REGION Network 138: Step[3090] : Job[21] Step End
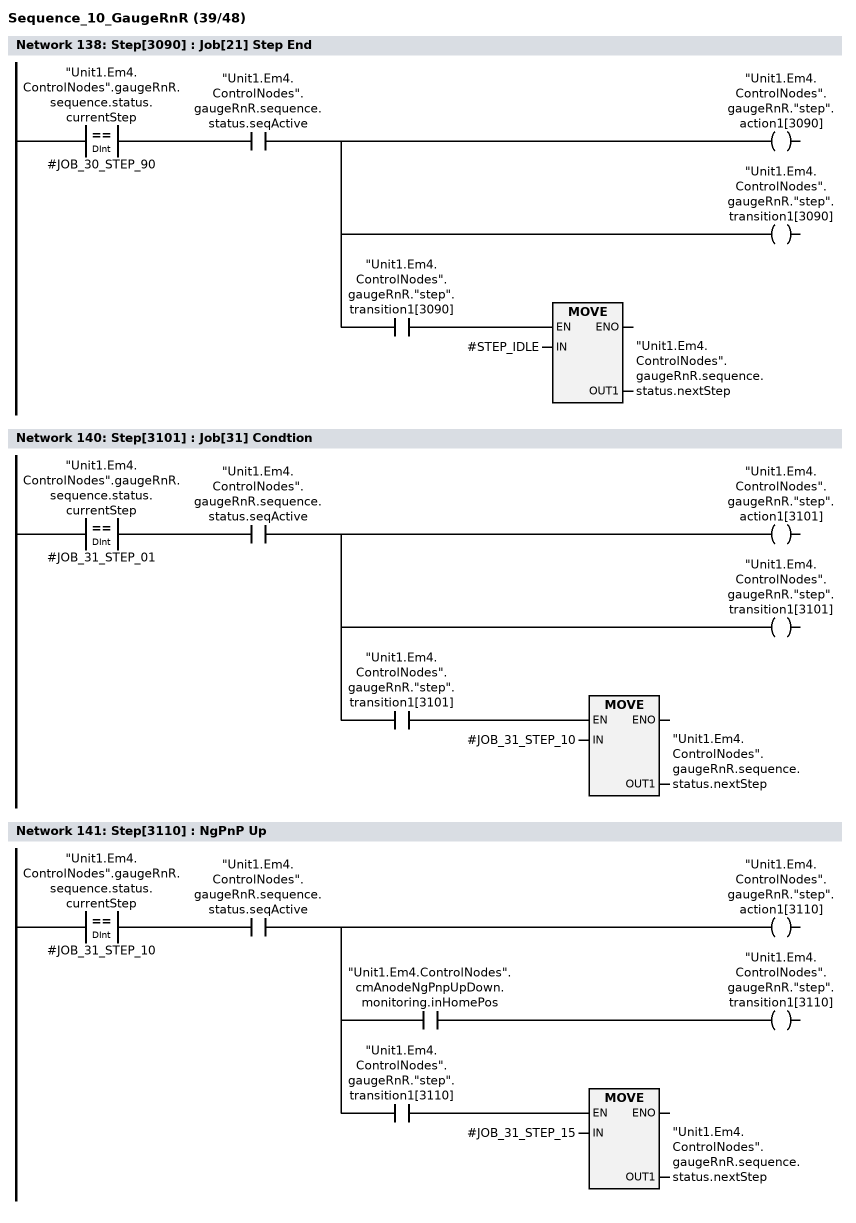
   RUNG wire#powerrail
      { S7_Templates := "SrcType := DInt" } EQ_Contact(in1 := "Unit1.Em4.ControlNodes".gaugeRnR.sequence.status.currentStep, in2 := #JOB_30_STEP_90)
      Contact( "Unit1.Em4.ControlNodes".gaugeRnR.sequence.status.seqActive )
      wire#w1
      Coil( "Unit1.Em4.ControlNodes".gaugeRnR."step".action1[3090] )
   END_RUNG
   RUNG wire#w1
      Coil( "Unit1.Em4.ControlNodes".gaugeRnR."step".transition1[3090] )
   END_RUNG
   RUNG wire#w1
      Contact( "Unit1.Em4.ControlNodes".gaugeRnR."step".transition1[3090] )
      Move(in := #STEP_IDLE, out1 => "Unit1.Em4.ControlNodes".gaugeRnR.sequence.status.nextStep)
   END_RUNG
   // the same network as SCL:
   "Unit1.Em4.ControlNodes".gaugeRnR."step".action1[3090] := ("Unit1.Em4.ControlNodes".gaugeRnR.sequence.status.currentStep = #JOB_30_STEP_90) AND "Unit1.Em4.ControlNodes".gaugeRnR.sequence.status.seqActive;
   "Unit1.Em4.ControlNodes".gaugeRnR."step".transition1[3090] := ("Unit1.Em4.ControlNodes".gaugeRnR.sequence.status.currentStep = #JOB_30_STEP_90) AND "Unit1.Em4.ControlNodes".gaugeRnR.sequence.status.seqActive;
   IF ("Unit1.Em4.ControlNodes".gaugeRnR.sequence.status.currentStep = #JOB_30_STEP_90) AND "Unit1.Em4.ControlNodes".gaugeRnR.sequence.status.seqActive AND "Unit1.Em4.ControlNodes".gaugeRnR."step".transition1[3090] THEN
       "Unit1.Em4.ControlNodes".gaugeRnR.sequence.status.nextStep := #STEP_IDLE;
   END_IF;
END_REGION

REGION Network 139: *************** JOB[31] NG PnP Load MasterPiece ************************
END_REGION

REGION Network 140: Step[3101] : Job[31] Condtion
   RUNG wire#powerrail
      { S7_Templates := "SrcType := DInt" } EQ_Contact(in1 := "Unit1.Em4.ControlNodes".gaugeRnR.sequence.status.currentStep, in2 := #JOB_31_STEP_01)
      Contact( "Unit1.Em4.ControlNodes".gaugeRnR.sequence.status.seqActive )
      wire#w1
      Coil( "Unit1.Em4.ControlNodes".gaugeRnR."step".action1[3101] )
   END_RUNG
   RUNG wire#w1
      Coil( "Unit1.Em4.ControlNodes".gaugeRnR."step".transition1[3101] )
   END_RUNG
   RUNG wire#w1
      Contact( "Unit1.Em4.ControlNodes".gaugeRnR."step".transition1[3101] )
      Move(in := #JOB_31_STEP_10, out1 => "Unit1.Em4.ControlNodes".gaugeRnR.sequence.status.nextStep)
   END_RUNG
   // the same network as SCL:
   "Unit1.Em4.ControlNodes".gaugeRnR."step".action1[3101] := ("Unit1.Em4.ControlNodes".gaugeRnR.sequence.status.currentStep = #JOB_31_STEP_01) AND "Unit1.Em4.ControlNodes".gaugeRnR.sequence.status.seqActive;
   "Unit1.Em4.ControlNodes".gaugeRnR."step".transition1[3101] := ("Unit1.Em4.ControlNodes".gaugeRnR.sequence.status.currentStep = #JOB_31_STEP_01) AND "Unit1.Em4.ControlNodes".gaugeRnR.sequence.status.seqActive;
   IF ("Unit1.Em4.ControlNodes".gaugeRnR.sequence.status.currentStep = #JOB_31_STEP_01) AND "Unit1.Em4.ControlNodes".gaugeRnR.sequence.status.seqActive AND "Unit1.Em4.ControlNodes".gaugeRnR."step".transition1[3101] THEN
       "Unit1.Em4.ControlNodes".gaugeRnR.sequence.status.nextStep := #JOB_31_STEP_10;
   END_IF;
END_REGION

REGION Network 141: Step[3110] : NgPnP Up
   RUNG wire#powerrail
      { S7_Templates := "SrcType := DInt" } EQ_Contact(in1 := "Unit1.Em4.ControlNodes".gaugeRnR.sequence.status.currentStep, in2 := #JOB_31_STEP_10)
      Contact( "Unit1.Em4.ControlNodes".gaugeRnR.sequence.status.seqActive )
      wire#w1
      Coil( "Unit1.Em4.ControlNodes".gaugeRnR."step".action1[3110] )
   END_RUNG
   RUNG wire#w1
      Contact( "Unit1.Em4.ControlNodes".cmAnodeNgPnpUpDown.monitoring.inHomePos )
      Coil( "Unit1.Em4.ControlNodes".gaugeRnR."step".transition1[3110] )
   END_RUNG
   RUNG wire#w1
      Contact( "Unit1.Em4.ControlNodes".gaugeRnR."step".transition1[3110] )
      Move(in := #JOB_31_STEP_15, out1 => "Unit1.Em4.ControlNodes".gaugeRnR.sequence.status.nextStep)
   END_RUNG
   // the same network as SCL:
   "Unit1.Em4.ControlNodes".gaugeRnR."step".action1[3110] := ("Unit1.Em4.ControlNodes".gaugeRnR.sequence.status.currentStep = #JOB_31_STEP_10) AND "Unit1.Em4.ControlNodes".gaugeRnR.sequence.status.seqActive;
   "Unit1.Em4.ControlNodes".gaugeRnR."step".transition1[3110] := ("Unit1.Em4.ControlNodes".gaugeRnR.sequence.status.currentStep = #JOB_31_STEP_10) AND "Unit1.Em4.ControlNodes".gaugeRnR.sequence.status.seqActive AND "Unit1.Em4.ControlNodes".cmAnodeNgPnpUpDown.monitoring.inHomePos;
   IF ("Unit1.Em4.ControlNodes".gaugeRnR.sequence.status.currentStep = #JOB_31_STEP_10) AND "Unit1.Em4.ControlNodes".gaugeRnR.sequence.status.seqActive AND "Unit1.Em4.ControlNodes".gaugeRnR."step".transition1[3110] THEN
       "Unit1.Em4.ControlNodes".gaugeRnR.sequence.status.nextStep := #JOB_31_STEP_15;
   END_IF;
END_REGION

REGION Network 142: Step[3115] : NgPnP 1st Forward
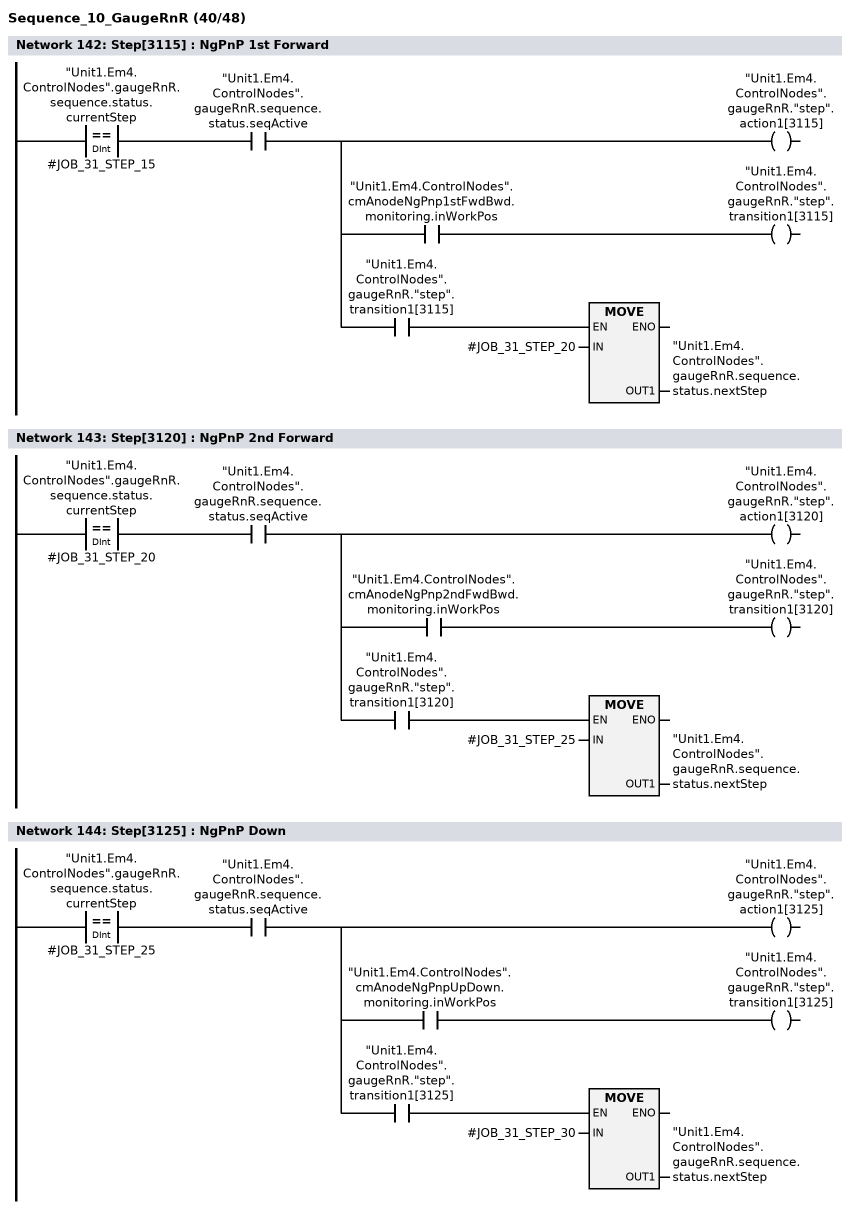
   RUNG wire#powerrail
      { S7_Templates := "SrcType := DInt" } EQ_Contact(in1 := "Unit1.Em4.ControlNodes".gaugeRnR.sequence.status.currentStep, in2 := #JOB_31_STEP_15)
      Contact( "Unit1.Em4.ControlNodes".gaugeRnR.sequence.status.seqActive )
      wire#w1
      Coil( "Unit1.Em4.ControlNodes".gaugeRnR."step".action1[3115] )
   END_RUNG
   RUNG wire#w1
      Contact( "Unit1.Em4.ControlNodes".cmAnodeNgPnp1stFwdBwd.monitoring.inWorkPos )
      Coil( "Unit1.Em4.ControlNodes".gaugeRnR."step".transition1[3115] )
   END_RUNG
   RUNG wire#w1
      Contact( "Unit1.Em4.ControlNodes".gaugeRnR."step".transition1[3115] )
      Move(in := #JOB_31_STEP_20, out1 => "Unit1.Em4.ControlNodes".gaugeRnR.sequence.status.nextStep)
   END_RUNG
   // the same network as SCL:
   "Unit1.Em4.ControlNodes".gaugeRnR."step".action1[3115] := ("Unit1.Em4.ControlNodes".gaugeRnR.sequence.status.currentStep = #JOB_31_STEP_15) AND "Unit1.Em4.ControlNodes".gaugeRnR.sequence.status.seqActive;
   "Unit1.Em4.ControlNodes".gaugeRnR."step".transition1[3115] := ("Unit1.Em4.ControlNodes".gaugeRnR.sequence.status.currentStep = #JOB_31_STEP_15) AND "Unit1.Em4.ControlNodes".gaugeRnR.sequence.status.seqActive AND "Unit1.Em4.ControlNodes".cmAnodeNgPnp1stFwdBwd.monitoring.inWorkPos;
   IF ("Unit1.Em4.ControlNodes".gaugeRnR.sequence.status.currentStep = #JOB_31_STEP_15) AND "Unit1.Em4.ControlNodes".gaugeRnR.sequence.status.seqActive AND "Unit1.Em4.ControlNodes".gaugeRnR."step".transition1[3115] THEN
       "Unit1.Em4.ControlNodes".gaugeRnR.sequence.status.nextStep := #JOB_31_STEP_20;
   END_IF;
END_REGION

REGION Network 143: Step[3120] : NgPnP 2nd Forward
   RUNG wire#powerrail
      { S7_Templates := "SrcType := DInt" } EQ_Contact(in1 := "Unit1.Em4.ControlNodes".gaugeRnR.sequence.status.currentStep, in2 := #JOB_31_STEP_20)
      Contact( "Unit1.Em4.ControlNodes".gaugeRnR.sequence.status.seqActive )
      wire#w1
      Coil( "Unit1.Em4.ControlNodes".gaugeRnR."step".action1[3120] )
   END_RUNG
   RUNG wire#w1
      Contact( "Unit1.Em4.ControlNodes".cmAnodeNgPnp2ndFwdBwd.monitoring.inWorkPos )
      Coil( "Unit1.Em4.ControlNodes".gaugeRnR."step".transition1[3120] )
   END_RUNG
   RUNG wire#w1
      Contact( "Unit1.Em4.ControlNodes".gaugeRnR."step".transition1[3120] )
      Move(in := #JOB_31_STEP_25, out1 => "Unit1.Em4.ControlNodes".gaugeRnR.sequence.status.nextStep)
   END_RUNG
   // the same network as SCL:
   "Unit1.Em4.ControlNodes".gaugeRnR."step".action1[3120] := ("Unit1.Em4.ControlNodes".gaugeRnR.sequence.status.currentStep = #JOB_31_STEP_20) AND "Unit1.Em4.ControlNodes".gaugeRnR.sequence.status.seqActive;
   "Unit1.Em4.ControlNodes".gaugeRnR."step".transition1[3120] := ("Unit1.Em4.ControlNodes".gaugeRnR.sequence.status.currentStep = #JOB_31_STEP_20) AND "Unit1.Em4.ControlNodes".gaugeRnR.sequence.status.seqActive AND "Unit1.Em4.ControlNodes".cmAnodeNgPnp2ndFwdBwd.monitoring.inWorkPos;
   IF ("Unit1.Em4.ControlNodes".gaugeRnR.sequence.status.currentStep = #JOB_31_STEP_20) AND "Unit1.Em4.ControlNodes".gaugeRnR.sequence.status.seqActive AND "Unit1.Em4.ControlNodes".gaugeRnR."step".transition1[3120] THEN
       "Unit1.Em4.ControlNodes".gaugeRnR.sequence.status.nextStep := #JOB_31_STEP_25;
   END_IF;
END_REGION

REGION Network 144: Step[3125] : NgPnP Down
   RUNG wire#powerrail
      { S7_Templates := "SrcType := DInt" } EQ_Contact(in1 := "Unit1.Em4.ControlNodes".gaugeRnR.sequence.status.currentStep, in2 := #JOB_31_STEP_25)
      Contact( "Unit1.Em4.ControlNodes".gaugeRnR.sequence.status.seqActive )
      wire#w1
      Coil( "Unit1.Em4.ControlNodes".gaugeRnR."step".action1[3125] )
   END_RUNG
   RUNG wire#w1
      Contact( "Unit1.Em4.ControlNodes".cmAnodeNgPnpUpDown.monitoring.inWorkPos )
      Coil( "Unit1.Em4.ControlNodes".gaugeRnR."step".transition1[3125] )
   END_RUNG
   RUNG wire#w1
      Contact( "Unit1.Em4.ControlNodes".gaugeRnR."step".transition1[3125] )
      Move(in := #JOB_31_STEP_30, out1 => "Unit1.Em4.ControlNodes".gaugeRnR.sequence.status.nextStep)
   END_RUNG
   // the same network as SCL:
   "Unit1.Em4.ControlNodes".gaugeRnR."step".action1[3125] := ("Unit1.Em4.ControlNodes".gaugeRnR.sequence.status.currentStep = #JOB_31_STEP_25) AND "Unit1.Em4.ControlNodes".gaugeRnR.sequence.status.seqActive;
   "Unit1.Em4.ControlNodes".gaugeRnR."step".transition1[3125] := ("Unit1.Em4.ControlNodes".gaugeRnR.sequence.status.currentStep = #JOB_31_STEP_25) AND "Unit1.Em4.ControlNodes".gaugeRnR.sequence.status.seqActive AND "Unit1.Em4.ControlNodes".cmAnodeNgPnpUpDown.monitoring.inWorkPos;
   IF ("Unit1.Em4.ControlNodes".gaugeRnR.sequence.status.currentStep = #JOB_31_STEP_25) AND "Unit1.Em4.ControlNodes".gaugeRnR.sequence.status.seqActive AND "Unit1.Em4.ControlNodes".gaugeRnR."step".transition1[3125] THEN
       "Unit1.Em4.ControlNodes".gaugeRnR.sequence.status.nextStep := #JOB_31_STEP_30;
   END_IF;
END_REGION

REGION Network 145: Step[3130] : AlignTable Vacuum Off
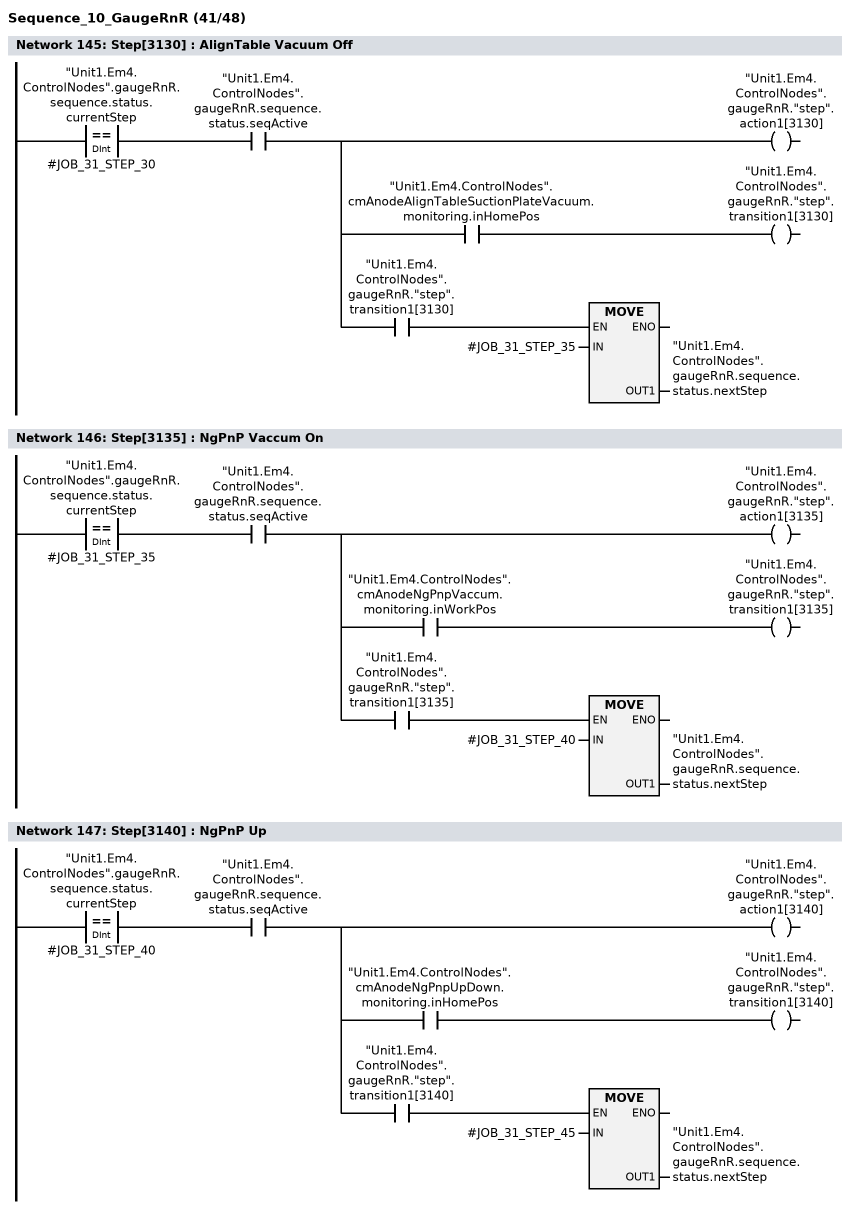
   RUNG wire#powerrail
      { S7_Templates := "SrcType := DInt" } EQ_Contact(in1 := "Unit1.Em4.ControlNodes".gaugeRnR.sequence.status.currentStep, in2 := #JOB_31_STEP_30)
      Contact( "Unit1.Em4.ControlNodes".gaugeRnR.sequence.status.seqActive )
      wire#w1
      Coil( "Unit1.Em4.ControlNodes".gaugeRnR."step".action1[3130] )
   END_RUNG
   RUNG wire#w1
      Contact( "Unit1.Em4.ControlNodes".cmAnodeAlignTableSuctionPlateVacuum.monitoring.inHomePos )
      Coil( "Unit1.Em4.ControlNodes".gaugeRnR."step".transition1[3130] )
   END_RUNG
   RUNG wire#w1
      Contact( "Unit1.Em4.ControlNodes".gaugeRnR."step".transition1[3130] )
      Move(in := #JOB_31_STEP_35, out1 => "Unit1.Em4.ControlNodes".gaugeRnR.sequence.status.nextStep)
   END_RUNG
   // the same network as SCL:
   "Unit1.Em4.ControlNodes".gaugeRnR."step".action1[3130] := ("Unit1.Em4.ControlNodes".gaugeRnR.sequence.status.currentStep = #JOB_31_STEP_30) AND "Unit1.Em4.ControlNodes".gaugeRnR.sequence.status.seqActive;
   "Unit1.Em4.ControlNodes".gaugeRnR."step".transition1[3130] := ("Unit1.Em4.ControlNodes".gaugeRnR.sequence.status.currentStep = #JOB_31_STEP_30) AND "Unit1.Em4.ControlNodes".gaugeRnR.sequence.status.seqActive AND "Unit1.Em4.ControlNodes".cmAnodeAlignTableSuctionPlateVacuum.monitoring.inHomePos;
   IF ("Unit1.Em4.ControlNodes".gaugeRnR.sequence.status.currentStep = #JOB_31_STEP_30) AND "Unit1.Em4.ControlNodes".gaugeRnR.sequence.status.seqActive AND "Unit1.Em4.ControlNodes".gaugeRnR."step".transition1[3130] THEN
       "Unit1.Em4.ControlNodes".gaugeRnR.sequence.status.nextStep := #JOB_31_STEP_35;
   END_IF;
END_REGION

REGION Network 146: Step[3135] : NgPnP Vaccum On
   RUNG wire#powerrail
      { S7_Templates := "SrcType := DInt" } EQ_Contact(in1 := "Unit1.Em4.ControlNodes".gaugeRnR.sequence.status.currentStep, in2 := #JOB_31_STEP_35)
      Contact( "Unit1.Em4.ControlNodes".gaugeRnR.sequence.status.seqActive )
      wire#w1
      Coil( "Unit1.Em4.ControlNodes".gaugeRnR."step".action1[3135] )
   END_RUNG
   RUNG wire#w1
      Contact( "Unit1.Em4.ControlNodes".cmAnodeNgPnpVaccum.monitoring.inWorkPos )
      Coil( "Unit1.Em4.ControlNodes".gaugeRnR."step".transition1[3135] )
   END_RUNG
   RUNG wire#w1
      Contact( "Unit1.Em4.ControlNodes".gaugeRnR."step".transition1[3135] )
      Move(in := #JOB_31_STEP_40, out1 => "Unit1.Em4.ControlNodes".gaugeRnR.sequence.status.nextStep)
   END_RUNG
   // the same network as SCL:
   "Unit1.Em4.ControlNodes".gaugeRnR."step".action1[3135] := ("Unit1.Em4.ControlNodes".gaugeRnR.sequence.status.currentStep = #JOB_31_STEP_35) AND "Unit1.Em4.ControlNodes".gaugeRnR.sequence.status.seqActive;
   "Unit1.Em4.ControlNodes".gaugeRnR."step".transition1[3135] := ("Unit1.Em4.ControlNodes".gaugeRnR.sequence.status.currentStep = #JOB_31_STEP_35) AND "Unit1.Em4.ControlNodes".gaugeRnR.sequence.status.seqActive AND "Unit1.Em4.ControlNodes".cmAnodeNgPnpVaccum.monitoring.inWorkPos;
   IF ("Unit1.Em4.ControlNodes".gaugeRnR.sequence.status.currentStep = #JOB_31_STEP_35) AND "Unit1.Em4.ControlNodes".gaugeRnR.sequence.status.seqActive AND "Unit1.Em4.ControlNodes".gaugeRnR."step".transition1[3135] THEN
       "Unit1.Em4.ControlNodes".gaugeRnR.sequence.status.nextStep := #JOB_31_STEP_40;
   END_IF;
END_REGION

REGION Network 147: Step[3140] : NgPnP Up
   RUNG wire#powerrail
      { S7_Templates := "SrcType := DInt" } EQ_Contact(in1 := "Unit1.Em4.ControlNodes".gaugeRnR.sequence.status.currentStep, in2 := #JOB_31_STEP_40)
      Contact( "Unit1.Em4.ControlNodes".gaugeRnR.sequence.status.seqActive )
      wire#w1
      Coil( "Unit1.Em4.ControlNodes".gaugeRnR."step".action1[3140] )
   END_RUNG
   RUNG wire#w1
      Contact( "Unit1.Em4.ControlNodes".cmAnodeNgPnpUpDown.monitoring.inHomePos )
      Coil( "Unit1.Em4.ControlNodes".gaugeRnR."step".transition1[3140] )
   END_RUNG
   RUNG wire#w1
      Contact( "Unit1.Em4.ControlNodes".gaugeRnR."step".transition1[3140] )
      Move(in := #JOB_31_STEP_45, out1 => "Unit1.Em4.ControlNodes".gaugeRnR.sequence.status.nextStep)
   END_RUNG
   // the same network as SCL:
   "Unit1.Em4.ControlNodes".gaugeRnR."step".action1[3140] := ("Unit1.Em4.ControlNodes".gaugeRnR.sequence.status.currentStep = #JOB_31_STEP_40) AND "Unit1.Em4.ControlNodes".gaugeRnR.sequence.status.seqActive;
   "Unit1.Em4.ControlNodes".gaugeRnR."step".transition1[3140] := ("Unit1.Em4.ControlNodes".gaugeRnR.sequence.status.currentStep = #JOB_31_STEP_40) AND "Unit1.Em4.ControlNodes".gaugeRnR.sequence.status.seqActive AND "Unit1.Em4.ControlNodes".cmAnodeNgPnpUpDown.monitoring.inHomePos;
   IF ("Unit1.Em4.ControlNodes".gaugeRnR.sequence.status.currentStep = #JOB_31_STEP_40) AND "Unit1.Em4.ControlNodes".gaugeRnR.sequence.status.seqActive AND "Unit1.Em4.ControlNodes".gaugeRnR."step".transition1[3140] THEN
       "Unit1.Em4.ControlNodes".gaugeRnR.sequence.status.nextStep := #JOB_31_STEP_45;
   END_IF;
END_REGION

REGION Network 148: Step[3145] : NgPnP 1st Backward
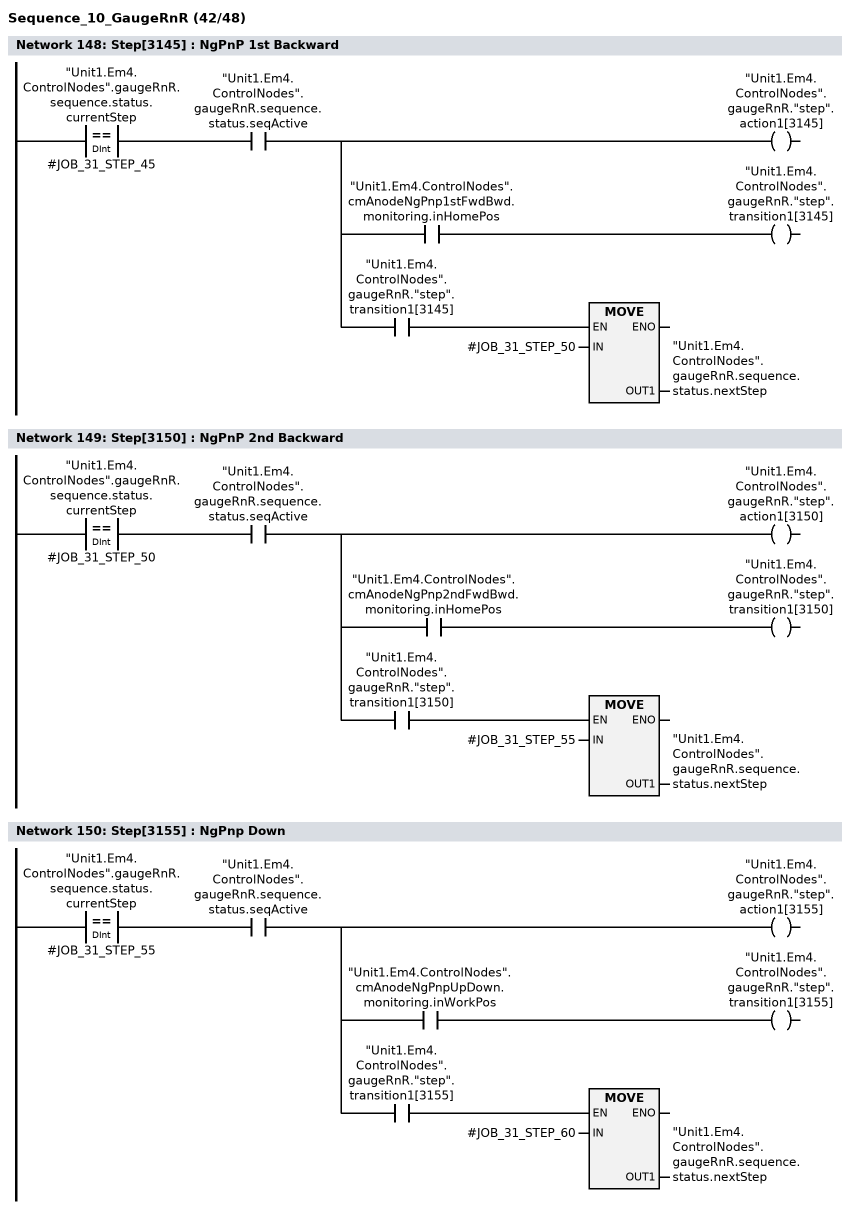
   RUNG wire#powerrail
      { S7_Templates := "SrcType := DInt" } EQ_Contact(in1 := "Unit1.Em4.ControlNodes".gaugeRnR.sequence.status.currentStep, in2 := #JOB_31_STEP_45)
      Contact( "Unit1.Em4.ControlNodes".gaugeRnR.sequence.status.seqActive )
      wire#w1
      Coil( "Unit1.Em4.ControlNodes".gaugeRnR."step".action1[3145] )
   END_RUNG
   RUNG wire#w1
      Contact( "Unit1.Em4.ControlNodes".cmAnodeNgPnp1stFwdBwd.monitoring.inHomePos )
      Coil( "Unit1.Em4.ControlNodes".gaugeRnR."step".transition1[3145] )
   END_RUNG
   RUNG wire#w1
      Contact( "Unit1.Em4.ControlNodes".gaugeRnR."step".transition1[3145] )
      Move(in := #JOB_31_STEP_50, out1 => "Unit1.Em4.ControlNodes".gaugeRnR.sequence.status.nextStep)
   END_RUNG
   // the same network as SCL:
   "Unit1.Em4.ControlNodes".gaugeRnR."step".action1[3145] := ("Unit1.Em4.ControlNodes".gaugeRnR.sequence.status.currentStep = #JOB_31_STEP_45) AND "Unit1.Em4.ControlNodes".gaugeRnR.sequence.status.seqActive;
   "Unit1.Em4.ControlNodes".gaugeRnR."step".transition1[3145] := ("Unit1.Em4.ControlNodes".gaugeRnR.sequence.status.currentStep = #JOB_31_STEP_45) AND "Unit1.Em4.ControlNodes".gaugeRnR.sequence.status.seqActive AND "Unit1.Em4.ControlNodes".cmAnodeNgPnp1stFwdBwd.monitoring.inHomePos;
   IF ("Unit1.Em4.ControlNodes".gaugeRnR.sequence.status.currentStep = #JOB_31_STEP_45) AND "Unit1.Em4.ControlNodes".gaugeRnR.sequence.status.seqActive AND "Unit1.Em4.ControlNodes".gaugeRnR."step".transition1[3145] THEN
       "Unit1.Em4.ControlNodes".gaugeRnR.sequence.status.nextStep := #JOB_31_STEP_50;
   END_IF;
END_REGION

REGION Network 149: Step[3150] : NgPnP 2nd Backward
   RUNG wire#powerrail
      { S7_Templates := "SrcType := DInt" } EQ_Contact(in1 := "Unit1.Em4.ControlNodes".gaugeRnR.sequence.status.currentStep, in2 := #JOB_31_STEP_50)
      Contact( "Unit1.Em4.ControlNodes".gaugeRnR.sequence.status.seqActive )
      wire#w1
      Coil( "Unit1.Em4.ControlNodes".gaugeRnR."step".action1[3150] )
   END_RUNG
   RUNG wire#w1
      Contact( "Unit1.Em4.ControlNodes".cmAnodeNgPnp2ndFwdBwd.monitoring.inHomePos )
      Coil( "Unit1.Em4.ControlNodes".gaugeRnR."step".transition1[3150] )
   END_RUNG
   RUNG wire#w1
      Contact( "Unit1.Em4.ControlNodes".gaugeRnR."step".transition1[3150] )
      Move(in := #JOB_31_STEP_55, out1 => "Unit1.Em4.ControlNodes".gaugeRnR.sequence.status.nextStep)
   END_RUNG
   // the same network as SCL:
   "Unit1.Em4.ControlNodes".gaugeRnR."step".action1[3150] := ("Unit1.Em4.ControlNodes".gaugeRnR.sequence.status.currentStep = #JOB_31_STEP_50) AND "Unit1.Em4.ControlNodes".gaugeRnR.sequence.status.seqActive;
   "Unit1.Em4.ControlNodes".gaugeRnR."step".transition1[3150] := ("Unit1.Em4.ControlNodes".gaugeRnR.sequence.status.currentStep = #JOB_31_STEP_50) AND "Unit1.Em4.ControlNodes".gaugeRnR.sequence.status.seqActive AND "Unit1.Em4.ControlNodes".cmAnodeNgPnp2ndFwdBwd.monitoring.inHomePos;
   IF ("Unit1.Em4.ControlNodes".gaugeRnR.sequence.status.currentStep = #JOB_31_STEP_50) AND "Unit1.Em4.ControlNodes".gaugeRnR.sequence.status.seqActive AND "Unit1.Em4.ControlNodes".gaugeRnR."step".transition1[3150] THEN
       "Unit1.Em4.ControlNodes".gaugeRnR.sequence.status.nextStep := #JOB_31_STEP_55;
   END_IF;
END_REGION

REGION Network 150: Step[3155] : NgPnp Down
   RUNG wire#powerrail
      { S7_Templates := "SrcType := DInt" } EQ_Contact(in1 := "Unit1.Em4.ControlNodes".gaugeRnR.sequence.status.currentStep, in2 := #JOB_31_STEP_55)
      Contact( "Unit1.Em4.ControlNodes".gaugeRnR.sequence.status.seqActive )
      wire#w1
      Coil( "Unit1.Em4.ControlNodes".gaugeRnR."step".action1[3155] )
   END_RUNG
   RUNG wire#w1
      Contact( "Unit1.Em4.ControlNodes".cmAnodeNgPnpUpDown.monitoring.inWorkPos )
      Coil( "Unit1.Em4.ControlNodes".gaugeRnR."step".transition1[3155] )
   END_RUNG
   RUNG wire#w1
      Contact( "Unit1.Em4.ControlNodes".gaugeRnR."step".transition1[3155] )
      Move(in := #JOB_31_STEP_60, out1 => "Unit1.Em4.ControlNodes".gaugeRnR.sequence.status.nextStep)
   END_RUNG
   // the same network as SCL:
   "Unit1.Em4.ControlNodes".gaugeRnR."step".action1[3155] := ("Unit1.Em4.ControlNodes".gaugeRnR.sequence.status.currentStep = #JOB_31_STEP_55) AND "Unit1.Em4.ControlNodes".gaugeRnR.sequence.status.seqActive;
   "Unit1.Em4.ControlNodes".gaugeRnR."step".transition1[3155] := ("Unit1.Em4.ControlNodes".gaugeRnR.sequence.status.currentStep = #JOB_31_STEP_55) AND "Unit1.Em4.ControlNodes".gaugeRnR.sequence.status.seqActive AND "Unit1.Em4.ControlNodes".cmAnodeNgPnpUpDown.monitoring.inWorkPos;
   IF ("Unit1.Em4.ControlNodes".gaugeRnR.sequence.status.currentStep = #JOB_31_STEP_55) AND "Unit1.Em4.ControlNodes".gaugeRnR.sequence.status.seqActive AND "Unit1.Em4.ControlNodes".gaugeRnR."step".transition1[3155] THEN
       "Unit1.Em4.ControlNodes".gaugeRnR.sequence.status.nextStep := #JOB_31_STEP_60;
   END_IF;
END_REGION

REGION Network 151: Step[3160] : NgPnP Vaccum Off
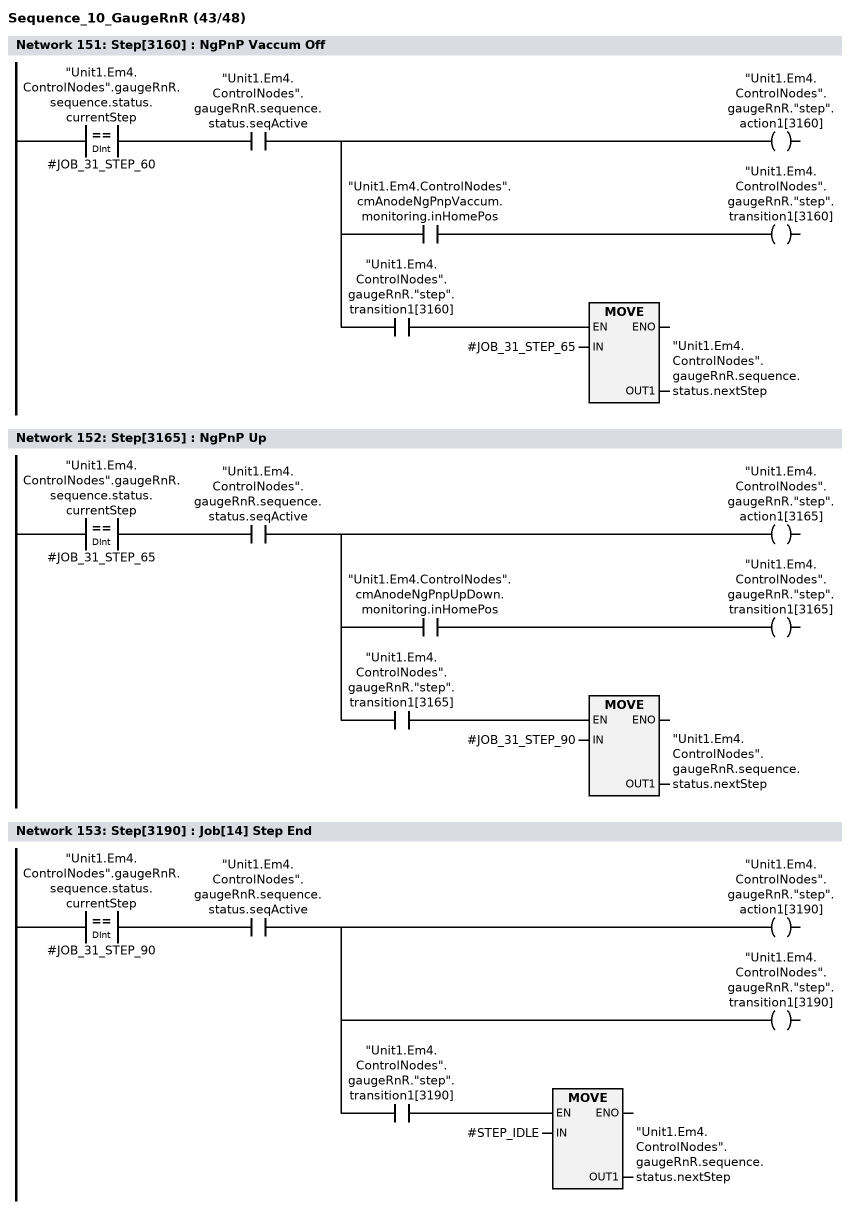
   RUNG wire#powerrail
      { S7_Templates := "SrcType := DInt" } EQ_Contact(in1 := "Unit1.Em4.ControlNodes".gaugeRnR.sequence.status.currentStep, in2 := #JOB_31_STEP_60)
      Contact( "Unit1.Em4.ControlNodes".gaugeRnR.sequence.status.seqActive )
      wire#w1
      Coil( "Unit1.Em4.ControlNodes".gaugeRnR."step".action1[3160] )
   END_RUNG
   RUNG wire#w1
      Contact( "Unit1.Em4.ControlNodes".cmAnodeNgPnpVaccum.monitoring.inHomePos )
      Coil( "Unit1.Em4.ControlNodes".gaugeRnR."step".transition1[3160] )
   END_RUNG
   RUNG wire#w1
      Contact( "Unit1.Em4.ControlNodes".gaugeRnR."step".transition1[3160] )
      Move(in := #JOB_31_STEP_65, out1 => "Unit1.Em4.ControlNodes".gaugeRnR.sequence.status.nextStep)
   END_RUNG
   // the same network as SCL:
   "Unit1.Em4.ControlNodes".gaugeRnR."step".action1[3160] := ("Unit1.Em4.ControlNodes".gaugeRnR.sequence.status.currentStep = #JOB_31_STEP_60) AND "Unit1.Em4.ControlNodes".gaugeRnR.sequence.status.seqActive;
   "Unit1.Em4.ControlNodes".gaugeRnR."step".transition1[3160] := ("Unit1.Em4.ControlNodes".gaugeRnR.sequence.status.currentStep = #JOB_31_STEP_60) AND "Unit1.Em4.ControlNodes".gaugeRnR.sequence.status.seqActive AND "Unit1.Em4.ControlNodes".cmAnodeNgPnpVaccum.monitoring.inHomePos;
   IF ("Unit1.Em4.ControlNodes".gaugeRnR.sequence.status.currentStep = #JOB_31_STEP_60) AND "Unit1.Em4.ControlNodes".gaugeRnR.sequence.status.seqActive AND "Unit1.Em4.ControlNodes".gaugeRnR."step".transition1[3160] THEN
       "Unit1.Em4.ControlNodes".gaugeRnR.sequence.status.nextStep := #JOB_31_STEP_65;
   END_IF;
END_REGION

REGION Network 152: Step[3165] : NgPnP Up
   RUNG wire#powerrail
      { S7_Templates := "SrcType := DInt" } EQ_Contact(in1 := "Unit1.Em4.ControlNodes".gaugeRnR.sequence.status.currentStep, in2 := #JOB_31_STEP_65)
      Contact( "Unit1.Em4.ControlNodes".gaugeRnR.sequence.status.seqActive )
      wire#w1
      Coil( "Unit1.Em4.ControlNodes".gaugeRnR."step".action1[3165] )
   END_RUNG
   RUNG wire#w1
      Contact( "Unit1.Em4.ControlNodes".cmAnodeNgPnpUpDown.monitoring.inHomePos )
      Coil( "Unit1.Em4.ControlNodes".gaugeRnR."step".transition1[3165] )
   END_RUNG
   RUNG wire#w1
      Contact( "Unit1.Em4.ControlNodes".gaugeRnR."step".transition1[3165] )
      Move(in := #JOB_31_STEP_90, out1 => "Unit1.Em4.ControlNodes".gaugeRnR.sequence.status.nextStep)
   END_RUNG
   // the same network as SCL:
   "Unit1.Em4.ControlNodes".gaugeRnR."step".action1[3165] := ("Unit1.Em4.ControlNodes".gaugeRnR.sequence.status.currentStep = #JOB_31_STEP_65) AND "Unit1.Em4.ControlNodes".gaugeRnR.sequence.status.seqActive;
   "Unit1.Em4.ControlNodes".gaugeRnR."step".transition1[3165] := ("Unit1.Em4.ControlNodes".gaugeRnR.sequence.status.currentStep = #JOB_31_STEP_65) AND "Unit1.Em4.ControlNodes".gaugeRnR.sequence.status.seqActive AND "Unit1.Em4.ControlNodes".cmAnodeNgPnpUpDown.monitoring.inHomePos;
   IF ("Unit1.Em4.ControlNodes".gaugeRnR.sequence.status.currentStep = #JOB_31_STEP_65) AND "Unit1.Em4.ControlNodes".gaugeRnR.sequence.status.seqActive AND "Unit1.Em4.ControlNodes".gaugeRnR."step".transition1[3165] THEN
       "Unit1.Em4.ControlNodes".gaugeRnR.sequence.status.nextStep := #JOB_31_STEP_90;
   END_IF;
END_REGION

REGION Network 153: Step[3190] : Job[14] Step End
   RUNG wire#powerrail
      { S7_Templates := "SrcType := DInt" } EQ_Contact(in1 := "Unit1.Em4.ControlNodes".gaugeRnR.sequence.status.currentStep, in2 := #JOB_31_STEP_90)
      Contact( "Unit1.Em4.ControlNodes".gaugeRnR.sequence.status.seqActive )
      wire#w1
      Coil( "Unit1.Em4.ControlNodes".gaugeRnR."step".action1[3190] )
   END_RUNG
   RUNG wire#w1
      Coil( "Unit1.Em4.ControlNodes".gaugeRnR."step".transition1[3190] )
   END_RUNG
   RUNG wire#w1
      Contact( "Unit1.Em4.ControlNodes".gaugeRnR."step".transition1[3190] )
      Move(in := #STEP_IDLE, out1 => "Unit1.Em4.ControlNodes".gaugeRnR.sequence.status.nextStep)
   END_RUNG
   // the same network as SCL:
   "Unit1.Em4.ControlNodes".gaugeRnR."step".action1[3190] := ("Unit1.Em4.ControlNodes".gaugeRnR.sequence.status.currentStep = #JOB_31_STEP_90) AND "Unit1.Em4.ControlNodes".gaugeRnR.sequence.status.seqActive;
   "Unit1.Em4.ControlNodes".gaugeRnR."step".transition1[3190] := ("Unit1.Em4.ControlNodes".gaugeRnR.sequence.status.currentStep = #JOB_31_STEP_90) AND "Unit1.Em4.ControlNodes".gaugeRnR.sequence.status.seqActive;
   IF ("Unit1.Em4.ControlNodes".gaugeRnR.sequence.status.currentStep = #JOB_31_STEP_90) AND "Unit1.Em4.ControlNodes".gaugeRnR.sequence.status.seqActive AND "Unit1.Em4.ControlNodes".gaugeRnR."step".transition1[3190] THEN
       "Unit1.Em4.ControlNodes".gaugeRnR.sequence.status.nextStep := #STEP_IDLE;
   END_IF;
END_REGION

REGION Network 154: *************** JOB[32] MainPnP2 Move AlignTable ************************
END_REGION

REGION Network 155: Step[3201] : Job[32] Condtion
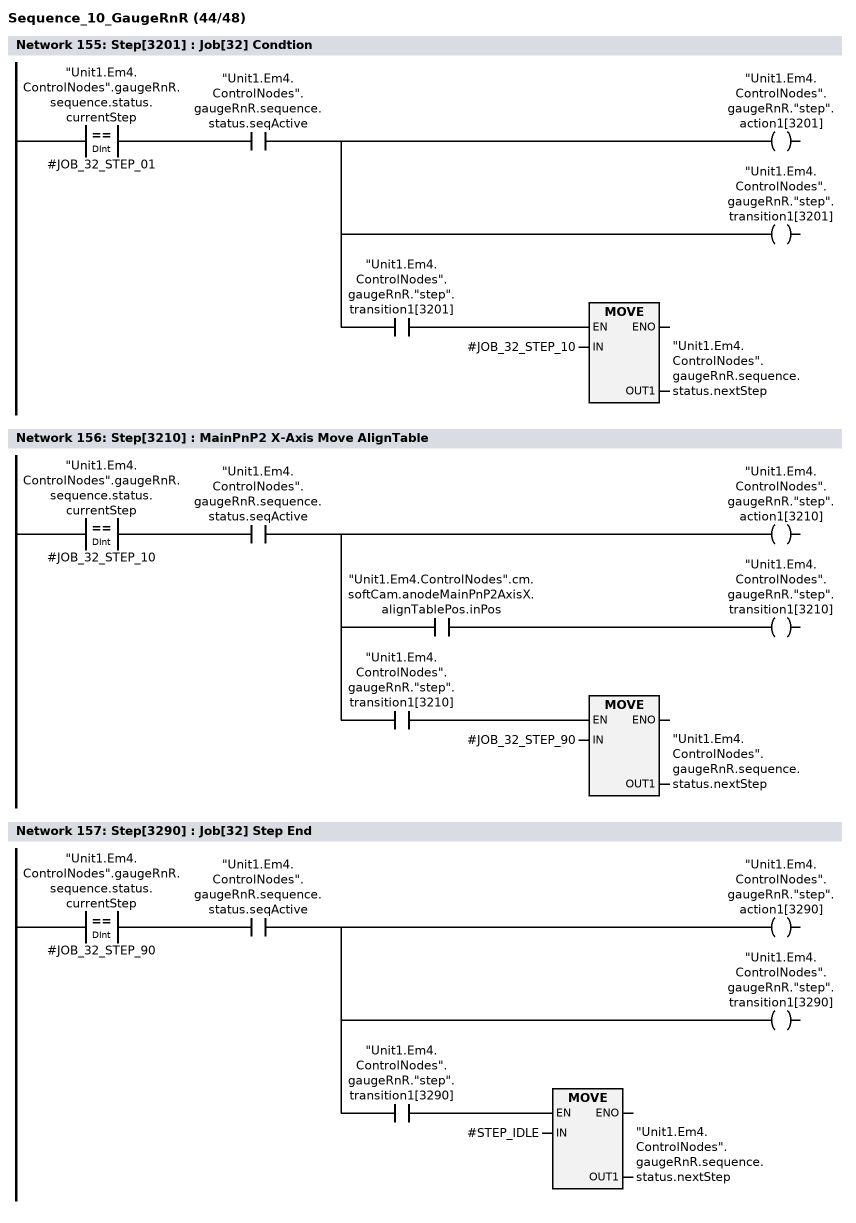
   RUNG wire#powerrail
      { S7_Templates := "SrcType := DInt" } EQ_Contact(in1 := "Unit1.Em4.ControlNodes".gaugeRnR.sequence.status.currentStep, in2 := #JOB_32_STEP_01)
      Contact( "Unit1.Em4.ControlNodes".gaugeRnR.sequence.status.seqActive )
      wire#w1
      Coil( "Unit1.Em4.ControlNodes".gaugeRnR."step".action1[3201] )
   END_RUNG
   RUNG wire#w1
      Coil( "Unit1.Em4.ControlNodes".gaugeRnR."step".transition1[3201] )
   END_RUNG
   RUNG wire#w1
      Contact( "Unit1.Em4.ControlNodes".gaugeRnR."step".transition1[3201] )
      Move(in := #JOB_32_STEP_10, out1 => "Unit1.Em4.ControlNodes".gaugeRnR.sequence.status.nextStep)
   END_RUNG
   // the same network as SCL:
   "Unit1.Em4.ControlNodes".gaugeRnR."step".action1[3201] := ("Unit1.Em4.ControlNodes".gaugeRnR.sequence.status.currentStep = #JOB_32_STEP_01) AND "Unit1.Em4.ControlNodes".gaugeRnR.sequence.status.seqActive;
   "Unit1.Em4.ControlNodes".gaugeRnR."step".transition1[3201] := ("Unit1.Em4.ControlNodes".gaugeRnR.sequence.status.currentStep = #JOB_32_STEP_01) AND "Unit1.Em4.ControlNodes".gaugeRnR.sequence.status.seqActive;
   IF ("Unit1.Em4.ControlNodes".gaugeRnR.sequence.status.currentStep = #JOB_32_STEP_01) AND "Unit1.Em4.ControlNodes".gaugeRnR.sequence.status.seqActive AND "Unit1.Em4.ControlNodes".gaugeRnR."step".transition1[3201] THEN
       "Unit1.Em4.ControlNodes".gaugeRnR.sequence.status.nextStep := #JOB_32_STEP_10;
   END_IF;
END_REGION

REGION Network 156: Step[3210] : MainPnP2 X-Axis Move AlignTable
   RUNG wire#powerrail
      { S7_Templates := "SrcType := DInt" } EQ_Contact(in1 := "Unit1.Em4.ControlNodes".gaugeRnR.sequence.status.currentStep, in2 := #JOB_32_STEP_10)
      Contact( "Unit1.Em4.ControlNodes".gaugeRnR.sequence.status.seqActive )
      wire#w1
      Coil( "Unit1.Em4.ControlNodes".gaugeRnR."step".action1[3210] )
   END_RUNG
   RUNG wire#w1
      Contact( "Unit1.Em4.ControlNodes".cm.softCam.anodeMainPnP2AxisX.alignTablePos.inPos )
      Coil( "Unit1.Em4.ControlNodes".gaugeRnR."step".transition1[3210] )
   END_RUNG
   RUNG wire#w1
      Contact( "Unit1.Em4.ControlNodes".gaugeRnR."step".transition1[3210] )
      Move(in := #JOB_32_STEP_90, out1 => "Unit1.Em4.ControlNodes".gaugeRnR.sequence.status.nextStep)
   END_RUNG
   // the same network as SCL:
   "Unit1.Em4.ControlNodes".gaugeRnR."step".action1[3210] := ("Unit1.Em4.ControlNodes".gaugeRnR.sequence.status.currentStep = #JOB_32_STEP_10) AND "Unit1.Em4.ControlNodes".gaugeRnR.sequence.status.seqActive;
   "Unit1.Em4.ControlNodes".gaugeRnR."step".transition1[3210] := ("Unit1.Em4.ControlNodes".gaugeRnR.sequence.status.currentStep = #JOB_32_STEP_10) AND "Unit1.Em4.ControlNodes".gaugeRnR.sequence.status.seqActive AND "Unit1.Em4.ControlNodes".cm.softCam.anodeMainPnP2AxisX.alignTablePos.inPos;
   IF ("Unit1.Em4.ControlNodes".gaugeRnR.sequence.status.currentStep = #JOB_32_STEP_10) AND "Unit1.Em4.ControlNodes".gaugeRnR.sequence.status.seqActive AND "Unit1.Em4.ControlNodes".gaugeRnR."step".transition1[3210] THEN
       "Unit1.Em4.ControlNodes".gaugeRnR.sequence.status.nextStep := #JOB_32_STEP_90;
   END_IF;
END_REGION

REGION Network 157: Step[3290] : Job[32] Step End
   RUNG wire#powerrail
      { S7_Templates := "SrcType := DInt" } EQ_Contact(in1 := "Unit1.Em4.ControlNodes".gaugeRnR.sequence.status.currentStep, in2 := #JOB_32_STEP_90)
      Contact( "Unit1.Em4.ControlNodes".gaugeRnR.sequence.status.seqActive )
      wire#w1
      Coil( "Unit1.Em4.ControlNodes".gaugeRnR."step".action1[3290] )
   END_RUNG
   RUNG wire#w1
      Coil( "Unit1.Em4.ControlNodes".gaugeRnR."step".transition1[3290] )
   END_RUNG
   RUNG wire#w1
      Contact( "Unit1.Em4.ControlNodes".gaugeRnR."step".transition1[3290] )
      Move(in := #STEP_IDLE, out1 => "Unit1.Em4.ControlNodes".gaugeRnR.sequence.status.nextStep)
   END_RUNG
   // the same network as SCL:
   "Unit1.Em4.ControlNodes".gaugeRnR."step".action1[3290] := ("Unit1.Em4.ControlNodes".gaugeRnR.sequence.status.currentStep = #JOB_32_STEP_90) AND "Unit1.Em4.ControlNodes".gaugeRnR.sequence.status.seqActive;
   "Unit1.Em4.ControlNodes".gaugeRnR."step".transition1[3290] := ("Unit1.Em4.ControlNodes".gaugeRnR.sequence.status.currentStep = #JOB_32_STEP_90) AND "Unit1.Em4.ControlNodes".gaugeRnR.sequence.status.seqActive;
   IF ("Unit1.Em4.ControlNodes".gaugeRnR.sequence.status.currentStep = #JOB_32_STEP_90) AND "Unit1.Em4.ControlNodes".gaugeRnR.sequence.status.seqActive AND "Unit1.Em4.ControlNodes".gaugeRnR."step".transition1[3290] THEN
       "Unit1.Em4.ControlNodes".gaugeRnR.sequence.status.nextStep := #STEP_IDLE;
   END_IF;
END_REGION

REGION Network 158: *************** JOB[33] AlignTable Move Wait ************************
END_REGION

REGION Network 159: Step[3301] : Job[33] Condtion
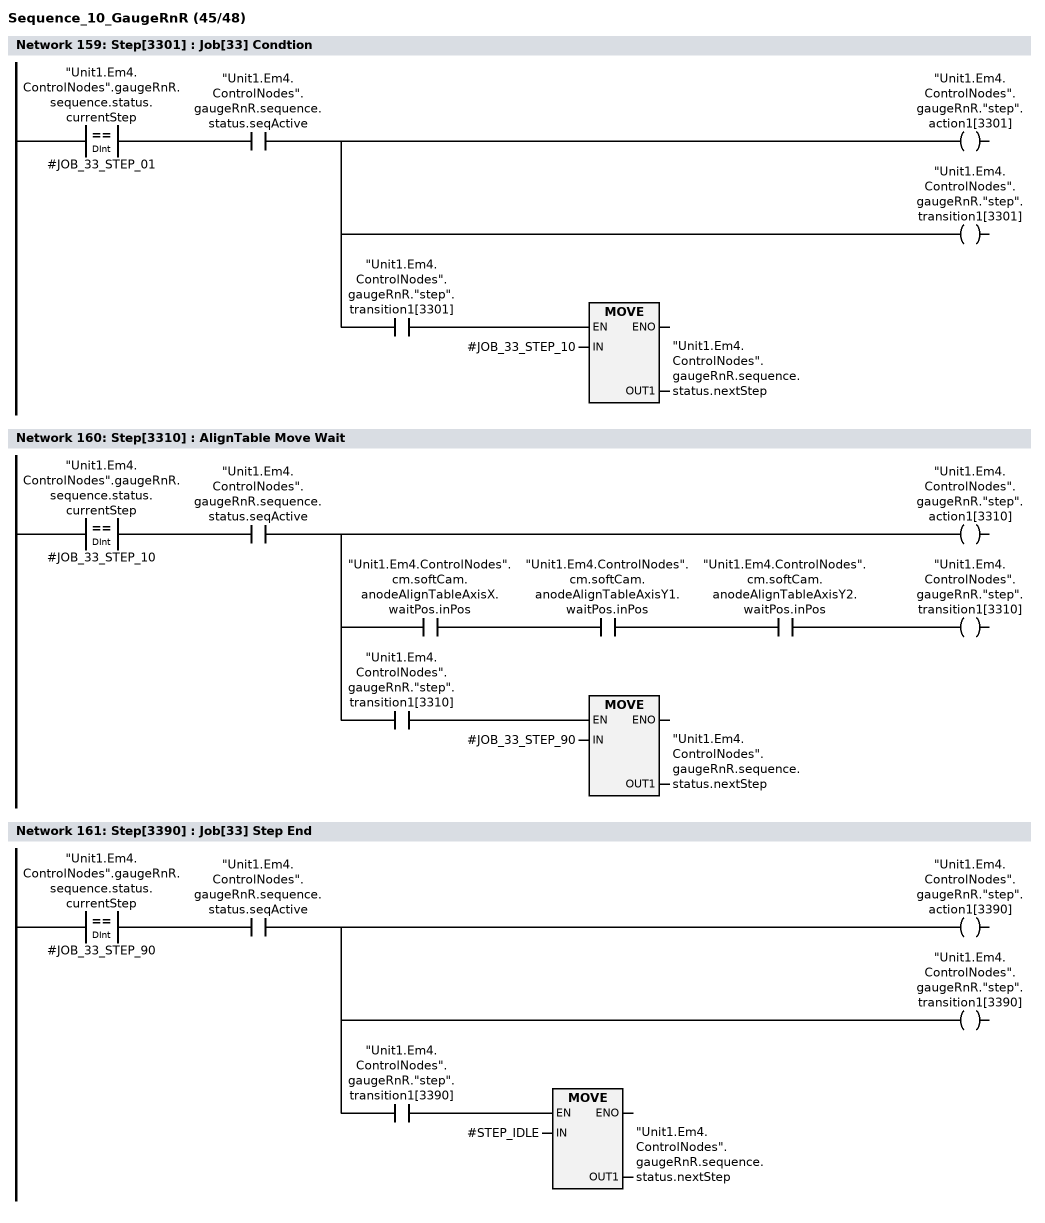
   RUNG wire#powerrail
      { S7_Templates := "SrcType := DInt" } EQ_Contact(in1 := "Unit1.Em4.ControlNodes".gaugeRnR.sequence.status.currentStep, in2 := #JOB_33_STEP_01)
      Contact( "Unit1.Em4.ControlNodes".gaugeRnR.sequence.status.seqActive )
      wire#w1
      Coil( "Unit1.Em4.ControlNodes".gaugeRnR."step".action1[3301] )
   END_RUNG
   RUNG wire#w1
      Coil( "Unit1.Em4.ControlNodes".gaugeRnR."step".transition1[3301] )
   END_RUNG
   RUNG wire#w1
      Contact( "Unit1.Em4.ControlNodes".gaugeRnR."step".transition1[3301] )
      Move(in := #JOB_33_STEP_10, out1 => "Unit1.Em4.ControlNodes".gaugeRnR.sequence.status.nextStep)
   END_RUNG
   // the same network as SCL:
   "Unit1.Em4.ControlNodes".gaugeRnR."step".action1[3301] := ("Unit1.Em4.ControlNodes".gaugeRnR.sequence.status.currentStep = #JOB_33_STEP_01) AND "Unit1.Em4.ControlNodes".gaugeRnR.sequence.status.seqActive;
   "Unit1.Em4.ControlNodes".gaugeRnR."step".transition1[3301] := ("Unit1.Em4.ControlNodes".gaugeRnR.sequence.status.currentStep = #JOB_33_STEP_01) AND "Unit1.Em4.ControlNodes".gaugeRnR.sequence.status.seqActive;
   IF ("Unit1.Em4.ControlNodes".gaugeRnR.sequence.status.currentStep = #JOB_33_STEP_01) AND "Unit1.Em4.ControlNodes".gaugeRnR.sequence.status.seqActive AND "Unit1.Em4.ControlNodes".gaugeRnR."step".transition1[3301] THEN
       "Unit1.Em4.ControlNodes".gaugeRnR.sequence.status.nextStep := #JOB_33_STEP_10;
   END_IF;
END_REGION

REGION Network 160: Step[3310] : AlignTable Move Wait
   RUNG wire#powerrail
      { S7_Templates := "SrcType := DInt" } EQ_Contact(in1 := "Unit1.Em4.ControlNodes".gaugeRnR.sequence.status.currentStep, in2 := #JOB_33_STEP_10)
      Contact( "Unit1.Em4.ControlNodes".gaugeRnR.sequence.status.seqActive )
      wire#w1
      Coil( "Unit1.Em4.ControlNodes".gaugeRnR."step".action1[3310] )
   END_RUNG
   RUNG wire#w1
      Contact( "Unit1.Em4.ControlNodes".cm.softCam.anodeAlignTableAxisX.waitPos.inPos )
      Contact( "Unit1.Em4.ControlNodes".cm.softCam.anodeAlignTableAxisY1.waitPos.inPos )
      Contact( "Unit1.Em4.ControlNodes".cm.softCam.anodeAlignTableAxisY2.waitPos.inPos )
      Coil( "Unit1.Em4.ControlNodes".gaugeRnR."step".transition1[3310] )
   END_RUNG
   RUNG wire#w1
      Contact( "Unit1.Em4.ControlNodes".gaugeRnR."step".transition1[3310] )
      Move(in := #JOB_33_STEP_90, out1 => "Unit1.Em4.ControlNodes".gaugeRnR.sequence.status.nextStep)
   END_RUNG
   // the same network as SCL:
   "Unit1.Em4.ControlNodes".gaugeRnR."step".action1[3310] := ("Unit1.Em4.ControlNodes".gaugeRnR.sequence.status.currentStep = #JOB_33_STEP_10) AND "Unit1.Em4.ControlNodes".gaugeRnR.sequence.status.seqActive;
   "Unit1.Em4.ControlNodes".gaugeRnR."step".transition1[3310] := ("Unit1.Em4.ControlNodes".gaugeRnR.sequence.status.currentStep = #JOB_33_STEP_10) AND "Unit1.Em4.ControlNodes".gaugeRnR.sequence.status.seqActive AND "Unit1.Em4.ControlNodes".cm.softCam.anodeAlignTableAxisX.waitPos.inPos AND "Unit1.Em4.ControlNodes".cm.softCam.anodeAlignTableAxisY1.waitPos.inPos AND "Unit1.Em4.ControlNodes".cm.softCam.anodeAlignTableAxisY2.waitPos.inPos;
   IF ("Unit1.Em4.ControlNodes".gaugeRnR.sequence.status.currentStep = #JOB_33_STEP_10) AND "Unit1.Em4.ControlNodes".gaugeRnR.sequence.status.seqActive AND "Unit1.Em4.ControlNodes".gaugeRnR."step".transition1[3310] THEN
       "Unit1.Em4.ControlNodes".gaugeRnR.sequence.status.nextStep := #JOB_33_STEP_90;
   END_IF;
END_REGION

REGION Network 161: Step[3390] : Job[33] Step End
   RUNG wire#powerrail
      { S7_Templates := "SrcType := DInt" } EQ_Contact(in1 := "Unit1.Em4.ControlNodes".gaugeRnR.sequence.status.currentStep, in2 := #JOB_33_STEP_90)
      Contact( "Unit1.Em4.ControlNodes".gaugeRnR.sequence.status.seqActive )
      wire#w1
      Coil( "Unit1.Em4.ControlNodes".gaugeRnR."step".action1[3390] )
   END_RUNG
   RUNG wire#w1
      Coil( "Unit1.Em4.ControlNodes".gaugeRnR."step".transition1[3390] )
   END_RUNG
   RUNG wire#w1
      Contact( "Unit1.Em4.ControlNodes".gaugeRnR."step".transition1[3390] )
      Move(in := #STEP_IDLE, out1 => "Unit1.Em4.ControlNodes".gaugeRnR.sequence.status.nextStep)
   END_RUNG
   // the same network as SCL:
   "Unit1.Em4.ControlNodes".gaugeRnR."step".action1[3390] := ("Unit1.Em4.ControlNodes".gaugeRnR.sequence.status.currentStep = #JOB_33_STEP_90) AND "Unit1.Em4.ControlNodes".gaugeRnR.sequence.status.seqActive;
   "Unit1.Em4.ControlNodes".gaugeRnR."step".transition1[3390] := ("Unit1.Em4.ControlNodes".gaugeRnR.sequence.status.currentStep = #JOB_33_STEP_90) AND "Unit1.Em4.ControlNodes".gaugeRnR.sequence.status.seqActive;
   IF ("Unit1.Em4.ControlNodes".gaugeRnR.sequence.status.currentStep = #JOB_33_STEP_90) AND "Unit1.Em4.ControlNodes".gaugeRnR.sequence.status.seqActive AND "Unit1.Em4.ControlNodes".gaugeRnR."step".transition1[3390] THEN
       "Unit1.Em4.ControlNodes".gaugeRnR.sequence.status.nextStep := #STEP_IDLE;
   END_IF;
END_REGION

REGION Network 162: *************** JOB[39] Common GugeRnR Complete ************************
END_REGION

REGION Network 163: Step[3901] : Job[39] Condtion
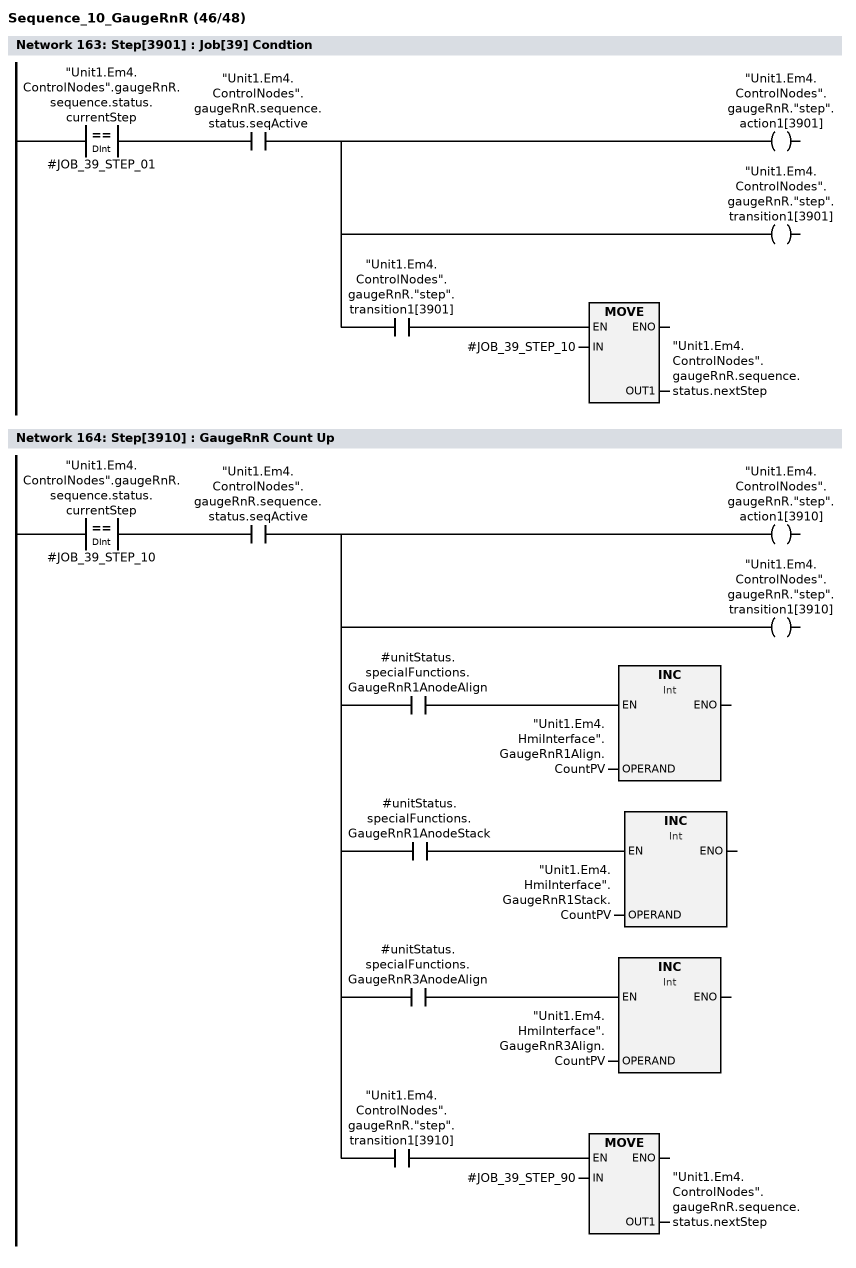
   RUNG wire#powerrail
      { S7_Templates := "SrcType := DInt" } EQ_Contact(in1 := "Unit1.Em4.ControlNodes".gaugeRnR.sequence.status.currentStep, in2 := #JOB_39_STEP_01)
      Contact( "Unit1.Em4.ControlNodes".gaugeRnR.sequence.status.seqActive )
      wire#w1
      Coil( "Unit1.Em4.ControlNodes".gaugeRnR."step".action1[3901] )
   END_RUNG
   RUNG wire#w1
      Coil( "Unit1.Em4.ControlNodes".gaugeRnR."step".transition1[3901] )
   END_RUNG
   RUNG wire#w1
      Contact( "Unit1.Em4.ControlNodes".gaugeRnR."step".transition1[3901] )
      Move(in := #JOB_39_STEP_10, out1 => "Unit1.Em4.ControlNodes".gaugeRnR.sequence.status.nextStep)
   END_RUNG
   // the same network as SCL:
   "Unit1.Em4.ControlNodes".gaugeRnR."step".action1[3901] := ("Unit1.Em4.ControlNodes".gaugeRnR.sequence.status.currentStep = #JOB_39_STEP_01) AND "Unit1.Em4.ControlNodes".gaugeRnR.sequence.status.seqActive;
   "Unit1.Em4.ControlNodes".gaugeRnR."step".transition1[3901] := ("Unit1.Em4.ControlNodes".gaugeRnR.sequence.status.currentStep = #JOB_39_STEP_01) AND "Unit1.Em4.ControlNodes".gaugeRnR.sequence.status.seqActive;
   IF ("Unit1.Em4.ControlNodes".gaugeRnR.sequence.status.currentStep = #JOB_39_STEP_01) AND "Unit1.Em4.ControlNodes".gaugeRnR.sequence.status.seqActive AND "Unit1.Em4.ControlNodes".gaugeRnR."step".transition1[3901] THEN
       "Unit1.Em4.ControlNodes".gaugeRnR.sequence.status.nextStep := #JOB_39_STEP_10;
   END_IF;
END_REGION

REGION Network 164: Step[3910] : GaugeRnR Count Up
   RUNG wire#powerrail
      { S7_Templates := "SrcType := DInt" } EQ_Contact(in1 := "Unit1.Em4.ControlNodes".gaugeRnR.sequence.status.currentStep, in2 := #JOB_39_STEP_10)
      Contact( "Unit1.Em4.ControlNodes".gaugeRnR.sequence.status.seqActive )
      wire#w1
      Coil( "Unit1.Em4.ControlNodes".gaugeRnR."step".action1[3910] )
   END_RUNG
   RUNG wire#w1
      Coil( "Unit1.Em4.ControlNodes".gaugeRnR."step".transition1[3910] )
   END_RUNG
   RUNG wire#w1
      Contact( #unitStatus.specialFunctions.GaugeRnR1AnodeAlign )
      { S7_Templates := "DestType := Int" } Inc( "Unit1.Em4.HmiInterface".GaugeRnR1Align.CountPV )
   END_RUNG
   RUNG wire#w1
      Contact( #unitStatus.specialFunctions.GaugeRnR1AnodeStack )
      { S7_Templates := "DestType := Int" } Inc( "Unit1.Em4.HmiInterface".GaugeRnR1Stack.CountPV )
   END_RUNG
   RUNG wire#w1
      Contact( #unitStatus.specialFunctions.GaugeRnR3AnodeAlign )
      { S7_Templates := "DestType := Int" } Inc( "Unit1.Em4.HmiInterface".GaugeRnR3Align.CountPV )
   END_RUNG
   RUNG wire#w1
      Contact( "Unit1.Em4.ControlNodes".gaugeRnR."step".transition1[3910] )
      Move(in := #JOB_39_STEP_90, out1 => "Unit1.Em4.ControlNodes".gaugeRnR.sequence.status.nextStep)
   END_RUNG
   // the same network as SCL:
   "Unit1.Em4.ControlNodes".gaugeRnR."step".action1[3910] := ("Unit1.Em4.ControlNodes".gaugeRnR.sequence.status.currentStep = #JOB_39_STEP_10) AND "Unit1.Em4.ControlNodes".gaugeRnR.sequence.status.seqActive;
   "Unit1.Em4.ControlNodes".gaugeRnR."step".transition1[3910] := ("Unit1.Em4.ControlNodes".gaugeRnR.sequence.status.currentStep = #JOB_39_STEP_10) AND "Unit1.Em4.ControlNodes".gaugeRnR.sequence.status.seqActive;
   IF ("Unit1.Em4.ControlNodes".gaugeRnR.sequence.status.currentStep = #JOB_39_STEP_10) AND "Unit1.Em4.ControlNodes".gaugeRnR.sequence.status.seqActive AND #unitStatus.specialFunctions.GaugeRnR1AnodeAlign THEN
       "Unit1.Em4.HmiInterface".GaugeRnR1Align.CountPV := "Unit1.Em4.HmiInterface".GaugeRnR1Align.CountPV + 1;
   END_IF;
   IF ("Unit1.Em4.ControlNodes".gaugeRnR.sequence.status.currentStep = #JOB_39_STEP_10) AND "Unit1.Em4.ControlNodes".gaugeRnR.sequence.status.seqActive AND #unitStatus.specialFunctions.GaugeRnR1AnodeStack THEN
       "Unit1.Em4.HmiInterface".GaugeRnR1Stack.CountPV := "Unit1.Em4.HmiInterface".GaugeRnR1Stack.CountPV + 1;
   END_IF;
   IF ("Unit1.Em4.ControlNodes".gaugeRnR.sequence.status.currentStep = #JOB_39_STEP_10) AND "Unit1.Em4.ControlNodes".gaugeRnR.sequence.status.seqActive AND #unitStatus.specialFunctions.GaugeRnR3AnodeAlign THEN
       "Unit1.Em4.HmiInterface".GaugeRnR3Align.CountPV := "Unit1.Em4.HmiInterface".GaugeRnR3Align.CountPV + 1;
   END_IF;
   IF ("Unit1.Em4.ControlNodes".gaugeRnR.sequence.status.currentStep = #JOB_39_STEP_10) AND "Unit1.Em4.ControlNodes".gaugeRnR.sequence.status.seqActive AND "Unit1.Em4.ControlNodes".gaugeRnR."step".transition1[3910] THEN
       "Unit1.Em4.ControlNodes".gaugeRnR.sequence.status.nextStep := #JOB_39_STEP_90;
   END_IF;
END_REGION

REGION Network 165: Step[3990] : Job[39] Step End
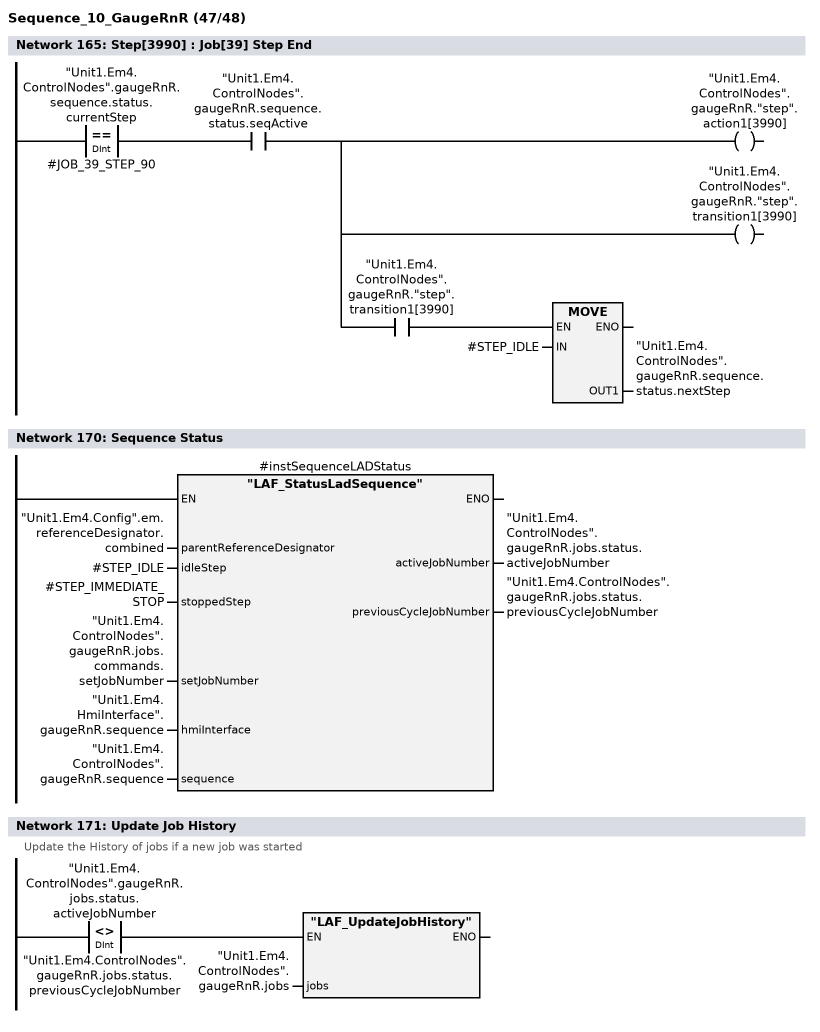
   RUNG wire#powerrail
      { S7_Templates := "SrcType := DInt" } EQ_Contact(in1 := "Unit1.Em4.ControlNodes".gaugeRnR.sequence.status.currentStep, in2 := #JOB_39_STEP_90)
      Contact( "Unit1.Em4.ControlNodes".gaugeRnR.sequence.status.seqActive )
      wire#w1
      Coil( "Unit1.Em4.ControlNodes".gaugeRnR."step".action1[3990] )
   END_RUNG
   RUNG wire#w1
      Coil( "Unit1.Em4.ControlNodes".gaugeRnR."step".transition1[3990] )
   END_RUNG
   RUNG wire#w1
      Contact( "Unit1.Em4.ControlNodes".gaugeRnR."step".transition1[3990] )
      Move(in := #STEP_IDLE, out1 => "Unit1.Em4.ControlNodes".gaugeRnR.sequence.status.nextStep)
   END_RUNG
   // the same network as SCL:
   "Unit1.Em4.ControlNodes".gaugeRnR."step".action1[3990] := ("Unit1.Em4.ControlNodes".gaugeRnR.sequence.status.currentStep = #JOB_39_STEP_90) AND "Unit1.Em4.ControlNodes".gaugeRnR.sequence.status.seqActive;
   "Unit1.Em4.ControlNodes".gaugeRnR."step".transition1[3990] := ("Unit1.Em4.ControlNodes".gaugeRnR.sequence.status.currentStep = #JOB_39_STEP_90) AND "Unit1.Em4.ControlNodes".gaugeRnR.sequence.status.seqActive;
   IF ("Unit1.Em4.ControlNodes".gaugeRnR.sequence.status.currentStep = #JOB_39_STEP_90) AND "Unit1.Em4.ControlNodes".gaugeRnR.sequence.status.seqActive AND "Unit1.Em4.ControlNodes".gaugeRnR."step".transition1[3990] THEN
       "Unit1.Em4.ControlNodes".gaugeRnR.sequence.status.nextStep := #STEP_IDLE;
   END_IF;
END_REGION

REGION Network 166: *************** IMMEDIATE STOP **************************
END_REGION

REGION Network 167: Immediate Stop
END_REGION

REGION Network 169: *************** Status updates **************************
END_REGION

REGION Network 170: Sequence Status
   RUNG wire#powerrail
      #instSequenceLADStatus(parentReferenceDesignator := "Unit1.Em4.Config".em.referenceDesignator.combined, idleStep := #STEP_IDLE, stoppedStep := #STEP_IMMEDIATE_STOP, setJobNumber := "Unit1.Em4.ControlNodes".gaugeRnR.jobs.commands.setJobNumber, hmiInterface := "Unit1.Em4.HmiInterface".gaugeRnR.sequence, sequence := "Unit1.Em4.ControlNodes".gaugeRnR.sequence, activeJobNumber => "Unit1.Em4.ControlNodes".gaugeRnR.jobs.status.activeJobNumber, previousCycleJobNumber => "Unit1.Em4.ControlNodes".gaugeRnR.jobs.status.previousCycleJobNumber)
   END_RUNG
   // the same network as SCL:
   #instSequenceLADStatus(parentReferenceDesignator := "Unit1.Em4.Config".em.referenceDesignator.combined,   // "LAF_StatusLadSequence"
                          idleStep := #STEP_IDLE,
                          stoppedStep := #STEP_IMMEDIATE_STOP,
                          setJobNumber := "Unit1.Em4.ControlNodes".gaugeRnR.jobs.commands.setJobNumber,
                          hmiInterface := "Unit1.Em4.HmiInterface".gaugeRnR.sequence,
                          sequence := "Unit1.Em4.ControlNodes".gaugeRnR.sequence,
                          activeJobNumber => "Unit1.Em4.ControlNodes".gaugeRnR.jobs.status.activeJobNumber,
                          previousCycleJobNumber => "Unit1.Em4.ControlNodes".gaugeRnR.jobs.status.previousCycleJobNumber);
END_REGION

REGION Network 171: Update Job History
   // Update the History of jobs if a new job was started
   RUNG wire#powerrail
      { S7_Templates := "SrcType := DInt" } NE_Contact(in1 := "Unit1.Em4.ControlNodes".gaugeRnR.jobs.status.activeJobNumber, in2 := "Unit1.Em4.ControlNodes".gaugeRnR.jobs.status.previousCycleJobNumber)
      "LAF_UpdateJobHistory"(jobs := "Unit1.Em4.ControlNodes".gaugeRnR.jobs)
   END_RUNG
   // the same network as SCL:
   IF "Unit1.Em4.ControlNodes".gaugeRnR.jobs.status.activeJobNumber <> "Unit1.Em4.ControlNodes".gaugeRnR.jobs.status.previousCycleJobNumber THEN
       "LAF_UpdateJobHistory"(jobs := "Unit1.Em4.ControlNodes".gaugeRnR.jobs);
   END_IF;
END_REGION

REGION Network 172: Output steps as String
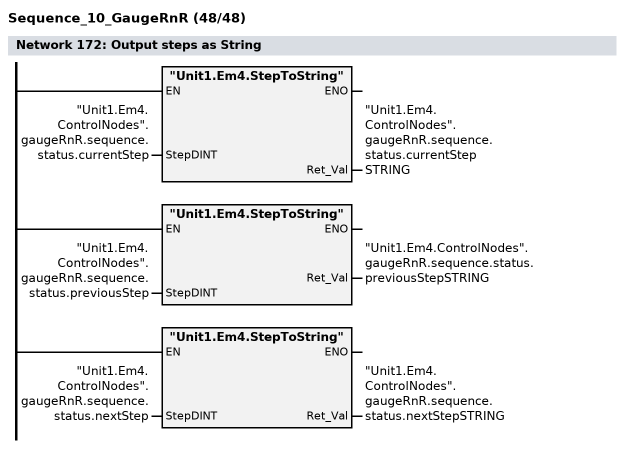
   RUNG wire#powerrail
      "Unit1.Em4.StepToString"(StepDINT := "Unit1.Em4.ControlNodes".gaugeRnR.sequence.status.currentStep, Ret_Val => "Unit1.Em4.ControlNodes".gaugeRnR.sequence.status.currentStepSTRING)
   END_RUNG
   RUNG wire#powerrail
      "Unit1.Em4.StepToString"(StepDINT := "Unit1.Em4.ControlNodes".gaugeRnR.sequence.status.previousStep, Ret_Val => "Unit1.Em4.ControlNodes".gaugeRnR.sequence.status.previousStepSTRING)
   END_RUNG
   RUNG wire#powerrail
      "Unit1.Em4.StepToString"(StepDINT := "Unit1.Em4.ControlNodes".gaugeRnR.sequence.status.nextStep, Ret_Val => "Unit1.Em4.ControlNodes".gaugeRnR.sequence.status.nextStepSTRING)
   END_RUNG
   // the same network as SCL:
   "Unit1.Em4.ControlNodes".gaugeRnR.sequence.status.currentStepSTRING := "Unit1.Em4.StepToString"(StepDINT := "Unit1.Em4.ControlNodes".gaugeRnR.sequence.status.currentStep);
   "Unit1.Em4.ControlNodes".gaugeRnR.sequence.status.previousStepSTRING := "Unit1.Em4.StepToString"(StepDINT := "Unit1.Em4.ControlNodes".gaugeRnR.sequence.status.previousStep);
   "Unit1.Em4.ControlNodes".gaugeRnR.sequence.status.nextStepSTRING := "Unit1.Em4.StepToString"(StepDINT := "Unit1.Em4.ControlNodes".gaugeRnR.sequence.status.nextStep);
END_REGION
END_FUNCTION_BLOCK
